FUNCTION_BLOCK TestModule_2
VAR_INPUT
	fbNextStationReleaseMaster : ReleaseMaster;
END_VAR
VAR_OUTPUT
END_VAR
VAR
END_VAR

fbNextStationReleaseMaster();

END_FUNCTION_BLOCK

(* stored: Version 1.1.0.1, ProductVersion 3.1.4024.2
   POU TestModule_2: Id {a7b992a4-5e40-4c2d-878b-802603a9aeaa}, SpecialFunc None *)
